# EPICS autosave request: galilDmc30017App/Db/galil_dmc30017_digital_out.req
# The files listed here are located at <GALIL support top>/GalilSup/Db
# as they are provided by the Galil Support Module

# All 4 Digital output bits
file "galil_digital_out_bit.req" P=$(P), R=$(DIG_OUT0)
file "galil_digital_out_bit.req" P=$(P), R=$(DIG_OUT1)
file "galil_digital_out_bit.req" P=$(P), R=$(DIG_OUT2)
file "galil_digital_out_bit.req" P=$(P), R=$(DIG_OUT3)
